INTERFACE I_ErrorAddedEvent EXTENDS I_Event

PROPERTY PUBLIC Target : I_Error
GET
END_GET
END_PROPERTY

END_INTERFACE

(* stored: Version 1.1.0.1, ProductVersion 3.1.4024.12
   Itf I_ErrorAddedEvent: Id {08a8faaf-cc56-0deb-204e-ea3cc40f76e7}
   Property Target: Id {9891ecd7-4ffb-01cb-0e25-f7863c3091df}
   Get Get: Id {083afae4-be20-0091-31ac-e587bd138cc5} *)
